TYPE ST_IvekCommandBits :
STRUCT
    // P010 Commands

    // Maintained command
    nMotionEnableBit      : USINT := 0;

    // Pulse commands
    nStopAllBit           : USINT := 1;
    nStartProductionBit   : USINT := 2;
    nStartFluidicBit      : USINT := 3;
    nStartReferenceBit    : USINT := 4;
    nClearFaultBit        : USINT := 5;
    nClearAlertBit        : USINT := 6;
    nStartLoadBit         : USINT := 7;

END_STRUCT
END_TYPE

(* stored: Version 1.1.0.1, ProductVersion 3.1.4026.18
   DUT ST_IvekCommandBits: Id {f78fb8cb-ad64-4e90-bf6e-f4552c1d9bc4} *)
